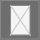
VISUALIZATION VISU_ButtonHome  // 40x40
    RoundedRectangle (0,0 40x40)
        OnMouseClick: change screen: VISU_Main
    Image (10,5 20x30), image: house_w
        OnMouseClick: change screen: VISU_Main
END_VISUALIZATION

(* stored: Version 1.1.0.1, ProductVersion 3.1.4024.11
   Visu VISU_ButtonHome: Id {a304afd2-8f89-4152-862a-bddad0d17b59} *)
